FUNCTION_BLOCK EA_RightPublishSubscribeAdapter
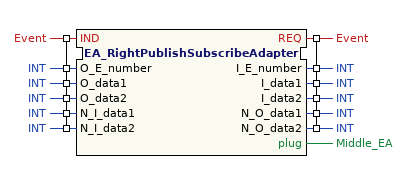
  EVENT_INPUT
    IND WITH O_E_number, O_data1, O_data2, N_I_data1, N_I_data2;
  END_EVENT
  EVENT_OUTPUT
    REQ WITH I_E_number, I_data1, I_data2, N_O_data1, N_O_data2;
  END_EVENT
  VAR_INPUT
    O_E_number : INT;
    O_data1 : INT;
    O_data2 : INT;
    N_I_data1 : INT;
    N_I_data2 : INT;
  END_VAR
  VAR_OUTPUT
    I_E_number : INT;
    I_data1 : INT;
    I_data2 : INT;
    N_O_data1 : INT;
    N_O_data2 : INT;
  END_VAR
  PLUGS
    plug : Middle_EA;
  END_PLUGS
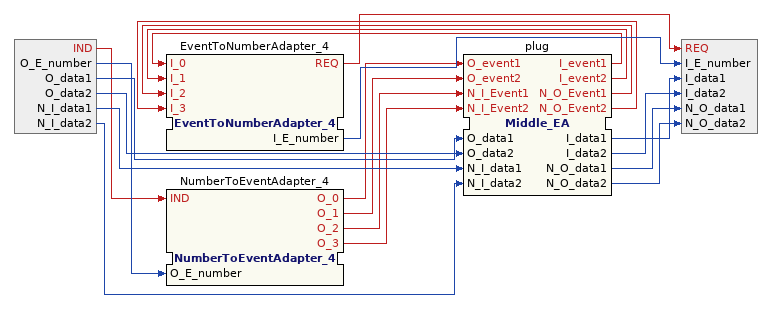
  FBS
    EventToNumberAdapter_4 : EventToNumberAdapter_4;
    NumberToEventAdapter_4 : NumberToEventAdapter_4;
  END_FBS
  EVENT_CONNECTIONS
    IND TO NumberToEventAdapter_4.IND;
    NumberToEventAdapter_4.O_0 TO plug.O_event1;
    NumberToEventAdapter_4.O_1 TO plug.O_event2;
    NumberToEventAdapter_4.O_2 TO plug.N_I_Event1;
    NumberToEventAdapter_4.O_3 TO plug.N_I_Event2;
    plug.I_event1 TO EventToNumberAdapter_4.I_0;
    plug.I_event2 TO EventToNumberAdapter_4.I_1;
    plug.N_O_Event1 TO EventToNumberAdapter_4.I_2;
    plug.N_O_Event2 TO EventToNumberAdapter_4.I_3;
    EventToNumberAdapter_4.REQ TO REQ;
  END_CONNECTIONS
  DATA_CONNECTIONS
    O_E_number TO NumberToEventAdapter_4.O_E_number;
    EventToNumberAdapter_4.I_E_number TO I_E_number;
    O_data1 TO plug.O_data1;
    O_data2 TO plug.O_data2;
    N_I_data1 TO plug.N_I_data1;
    N_I_data2 TO plug.N_I_data2;
    plug.I_data1 TO I_data1;
    plug.I_data2 TO I_data2;
    plug.N_O_data1 TO N_O_data1;
    plug.N_O_data2 TO N_O_data2;
  END_CONNECTIONS
END_FUNCTION_BLOCK
